{attribute addProperty BoxType "EL4032-0000-0016"}
{attribute addProperty Id "AO_Outputs_ChannelAT %Q*ARRAY[0..1] OF AO_Outputs_Channel_F57FA4F93240WcStateAT %I*WcState_28A8677510.1250InfoDataAT %I*InfoData_BC63D37F80100"}
{attribute addProperty CRC "3518482396"}
{attribute addProperty SizeInBites "113"}
{attribute addProperty SizeInBytes "14.125"}
TYPE EL4032_19A75BD9 :
STRUCT
	{attribute addProperty Name "AO_Outputs_Channel"}
	AO_Outputs_Channel : ARRAY[0..1] OF AO_Outputs_Channel_F57FA4F9;
	{attribute addProperty Name "WcState"}
	WcState : WcState_28A86775;
	{attribute addProperty Name "InfoData"}
	InfoData : InfoData_BC63D37F;
END_STRUCT
END_TYPE

(* stored: Version 1.2.0.0, ProductVersion 3.1.4024.9
   DUT EL4032_19A75BD9: Id {bd017138-db8e-43a1-aa59-f885d227c49e} *)
